// TIA Portal V19 export
TYPE "PII - AS5-AF2-FLX-G100"
   STRUCT
      "Process Data In - Mass Flow Rate" : Real;
      "Process Data In - Flow Velocity" : Real;
      "Process Data In - Volume" : Real;
      "Process Data In - Volumetric Flow Rate" : Real;
      "Process Data In - Mass" : Real;
      "Process Data In - Energy" : Real;
      "Process Data In - Temperature" : Real;
      "Process Data In - Pressure" : Real;
      "Port qualifier" : Byte;
   END_STRUCT;
END_TYPE
